{attribute 'qualified_only'}
{attribute 'strict'}
TYPE cPuckStatusEval :
(
	
	None := 0

) DINT;
END_TYPE

(* stored: Version 1.1.0.1, ProductVersion 3.1.4024.6
   DUT cPuckStatusEval: Id {e3578b67-131d-4ca2-8a9a-fe7d4c6decae} *)
